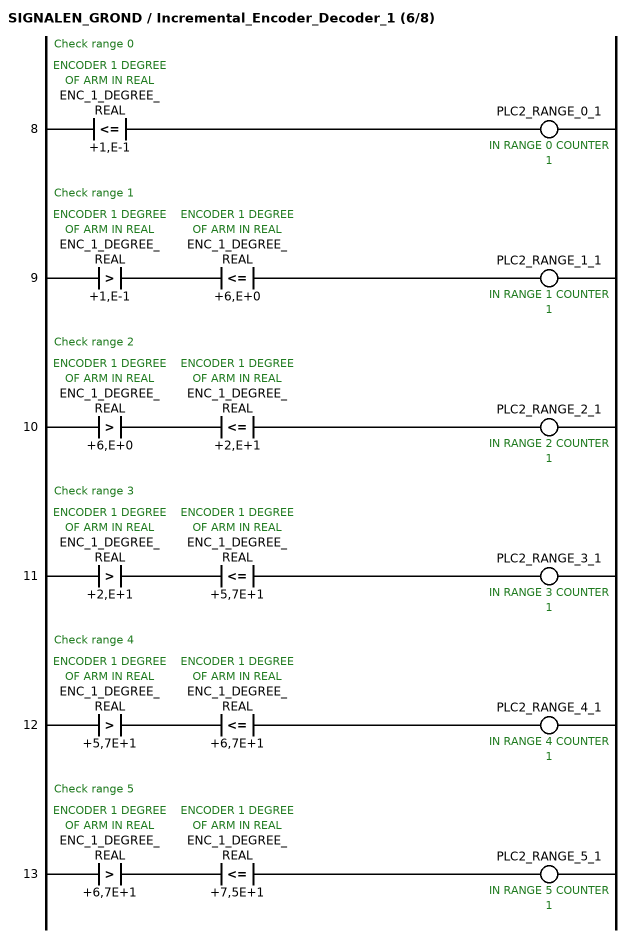
; [picture p325: SIGNALEN_GROND / Incremental_Encoder_Decoder_1, rungs 8-13]
; rung 8: Check range 0
LD<=F(332) ENC_1_DEGREE_REAL +1,E-1  ; ENCODER 1 DEGREE OF ARM IN REAL
OUT PLC2_RANGE_0_1  ; IN RANGE 0 COUNTER 1
; rung 9: Check range 1
LD>F(333) ENC_1_DEGREE_REAL +1,E-1  ; ENCODER 1 DEGREE OF ARM IN REAL
AND<=F(332) ENC_1_DEGREE_REAL +6,E+0  ; ENCODER 1 DEGREE OF ARM IN REAL
OUT PLC2_RANGE_1_1  ; IN RANGE 1 COUNTER 1
; rung 10: Check range 2
LD>F(333) ENC_1_DEGREE_REAL +6,E+0  ; ENCODER 1 DEGREE OF ARM IN REAL
AND<=F(332) ENC_1_DEGREE_REAL +2,E+1  ; ENCODER 1 DEGREE OF ARM IN REAL
OUT PLC2_RANGE_2_1  ; IN RANGE 2 COUNTER 1
; rung 11: Check range 3
LD>F(333) ENC_1_DEGREE_REAL +2,E+1  ; ENCODER 1 DEGREE OF ARM IN REAL
AND<=F(332) ENC_1_DEGREE_REAL +5,7E+1  ; ENCODER 1 DEGREE OF ARM IN REAL
OUT PLC2_RANGE_3_1  ; IN RANGE 3 COUNTER 1
; rung 12: Check range 4
LD>F(333) ENC_1_DEGREE_REAL +5,7E+1  ; ENCODER 1 DEGREE OF ARM IN REAL
AND<=F(332) ENC_1_DEGREE_REAL +6,7E+1  ; ENCODER 1 DEGREE OF ARM IN REAL
OUT PLC2_RANGE_4_1  ; IN RANGE 4 COUNTER 1
; rung 13: Check range 5
LD>F(333) ENC_1_DEGREE_REAL +6,7E+1  ; ENCODER 1 DEGREE OF ARM IN REAL
AND<=F(332) ENC_1_DEGREE_REAL +7,5E+1  ; ENCODER 1 DEGREE OF ARM IN REAL
OUT PLC2_RANGE_5_1  ; IN RANGE 5 COUNTER 1

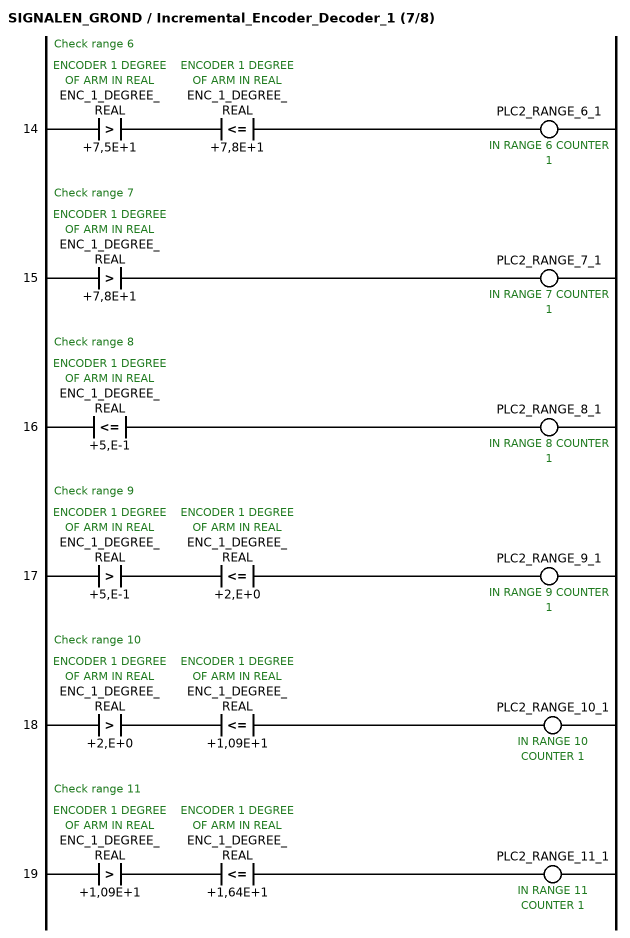
; rung 14: Check range 6
LD>F(333) ENC_1_DEGREE_REAL +7,5E+1  ; ENCODER 1 DEGREE OF ARM IN REAL
AND<=F(332) ENC_1_DEGREE_REAL +7,8E+1  ; ENCODER 1 DEGREE OF ARM IN REAL
OUT PLC2_RANGE_6_1  ; IN RANGE 6 COUNTER 1
; rung 15: Check range 7
LD>F(333) ENC_1_DEGREE_REAL +7,8E+1  ; ENCODER 1 DEGREE OF ARM IN REAL
OUT PLC2_RANGE_7_1  ; IN RANGE 7 COUNTER 1
; rung 16: Check range 8
LD<=F(332) ENC_1_DEGREE_REAL +5,E-1  ; ENCODER 1 DEGREE OF ARM IN REAL
OUT PLC2_RANGE_8_1  ; IN RANGE 8 COUNTER 1
; rung 17: Check range 9
LD>F(333) ENC_1_DEGREE_REAL +5,E-1  ; ENCODER 1 DEGREE OF ARM IN REAL
AND<=F(332) ENC_1_DEGREE_REAL +2,E+0  ; ENCODER 1 DEGREE OF ARM IN REAL
OUT PLC2_RANGE_9_1  ; IN RANGE 9 COUNTER 1
; rung 18: Check range 10
LD>F(333) ENC_1_DEGREE_REAL +2,E+0  ; ENCODER 1 DEGREE OF ARM IN REAL
AND<=F(332) ENC_1_DEGREE_REAL +1,09E+1  ; ENCODER 1 DEGREE OF ARM IN REAL
OUT PLC2_RANGE_10_1  ; IN RANGE 10 COUNTER 1
; rung 19: Check range 11
LD>F(333) ENC_1_DEGREE_REAL +1,09E+1  ; ENCODER 1 DEGREE OF ARM IN REAL
AND<=F(332) ENC_1_DEGREE_REAL +1,64E+1  ; ENCODER 1 DEGREE OF ARM IN REAL
OUT PLC2_RANGE_11_1  ; IN RANGE 11 COUNTER 1

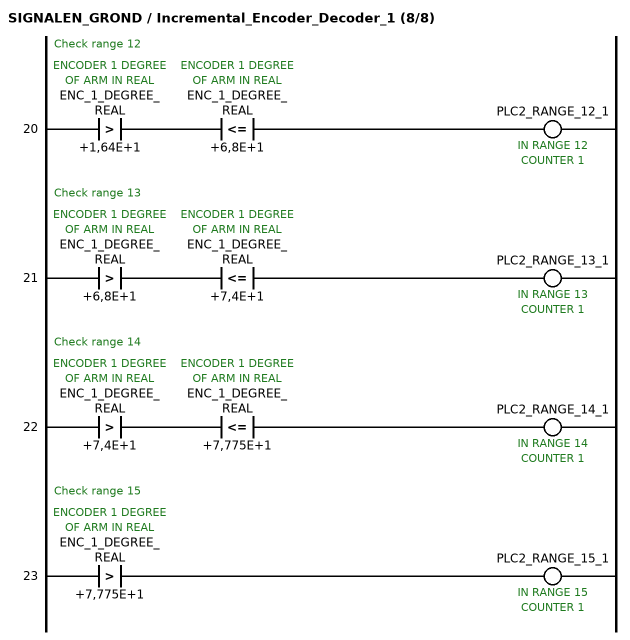
; rung 20: Check range 12
LD>F(333) ENC_1_DEGREE_REAL +1,64E+1  ; ENCODER 1 DEGREE OF ARM IN REAL
AND<=F(332) ENC_1_DEGREE_REAL +6,8E+1  ; ENCODER 1 DEGREE OF ARM IN REAL
OUT PLC2_RANGE_12_1  ; IN RANGE 12 COUNTER 1
; rung 21: Check range 13
LD>F(333) ENC_1_DEGREE_REAL +6,8E+1  ; ENCODER 1 DEGREE OF ARM IN REAL
AND<=F(332) ENC_1_DEGREE_REAL +7,4E+1  ; ENCODER 1 DEGREE OF ARM IN REAL
OUT PLC2_RANGE_13_1  ; IN RANGE 13 COUNTER 1
; rung 22: Check range 14
LD>F(333) ENC_1_DEGREE_REAL +7,4E+1  ; ENCODER 1 DEGREE OF ARM IN REAL
AND<=F(332) ENC_1_DEGREE_REAL +7,775E+1  ; ENCODER 1 DEGREE OF ARM IN REAL
OUT PLC2_RANGE_14_1  ; IN RANGE 14 COUNTER 1
; rung 23: Check range 15
LD>F(333) ENC_1_DEGREE_REAL +7,775E+1  ; ENCODER 1 DEGREE OF ARM IN REAL
OUT PLC2_RANGE_15_1  ; IN RANGE 15 COUNTER 1

### Section Incremental_Encoder_Decoder_2

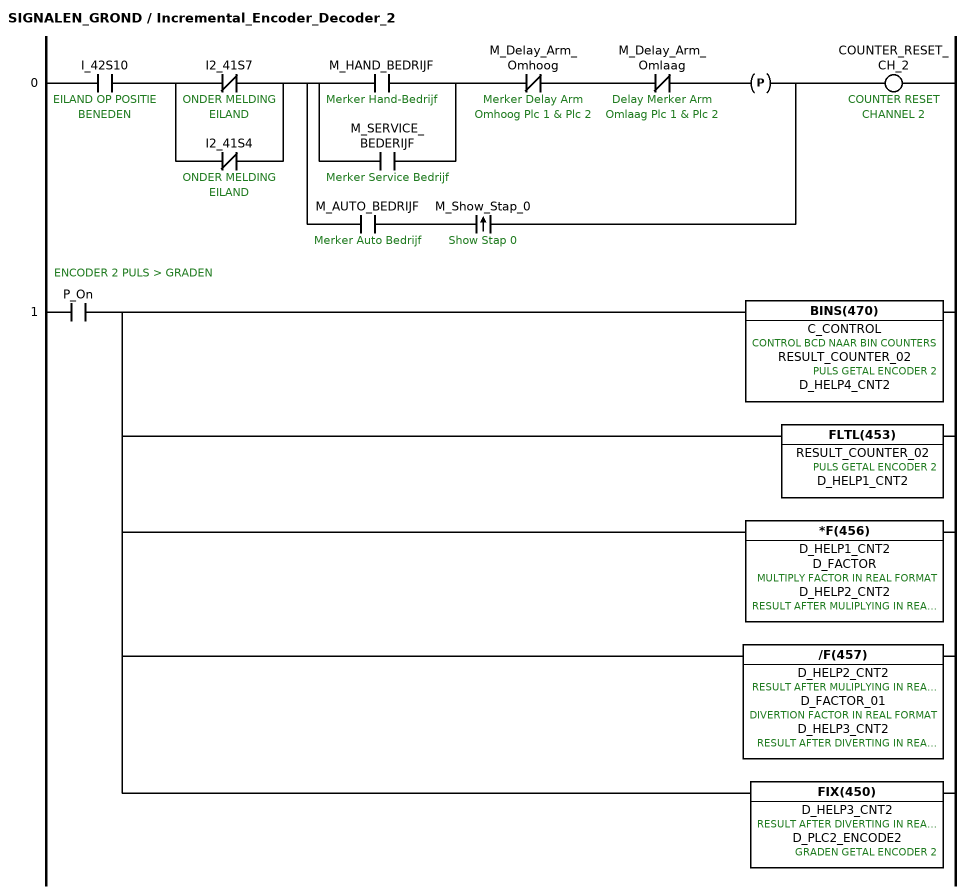
; rung 0
LD I_42S10  ; EILAND OP POSITIE BENEDEN
LDNOT I2_41S7  ; ONDER MELDING EILAND
ORNOT I2_41S4  ; ONDER MELDING EILAND
ANDLD
LD M_HAND_BEDRIJF  ; Merker Hand-Bedrijf
OR M_SERVICE_BEDERIJF  ; Merker Service Bedrijf
ANDNOT M_Delay_Arm_Omhoog  ; Merker Delay Arm Omhoog Plc 1 & Plc 2
ANDNOT M_Delay_Arm_Omlaag  ; Delay Merker Arm Omlaag Plc 1 & Plc 2
UP(521)
LD M_AUTO_BEDRIJF  ; Merker Auto Bedrijf
@AND M_Show_Stap_0  ; Show Stap 0
ORLD
ANDLD
OUT COUNTER_RESET_CH_2  ; COUNTER RESET CHANNEL 2
; rung 1: ENCODER 2 PULS > GRADEN
LD P_On
BINS(470) C_CONTROL RESULT_COUNTER_02 D_HELP4_CNT2  ; CONTROL BCD NAAR BIN COUNTERS, PULS GETAL ENCODER 2
FLTL(453) RESULT_COUNTER_02 D_HELP1_CNT2  ; PULS GETAL ENCODER 2
*F(456) D_HELP1_CNT2 D_FACTOR D_HELP2_CNT2  ; MULTIPLY FACTOR IN REAL FORMAT, RESULT AFTER MULIPLYING IN REAL FORMAT
/F(457) D_HELP2_CNT2 D_FACTOR_01 D_HELP3_CNT2  ; RESULT AFTER MULIPLYING IN REAL FORMAT, DIVERTION FACTOR IN REAL FORMAT, RESULT AFTER DIVERTING IN REAL FORMAT
FIX(450) D_HELP3_CNT2 D_PLC2_ENCODE2  ; RESULT AFTER DIVERTING IN REAL FORMAT, GRADEN GETAL ENCODER 2

### Section Absolute_Encoder_Decoder_3

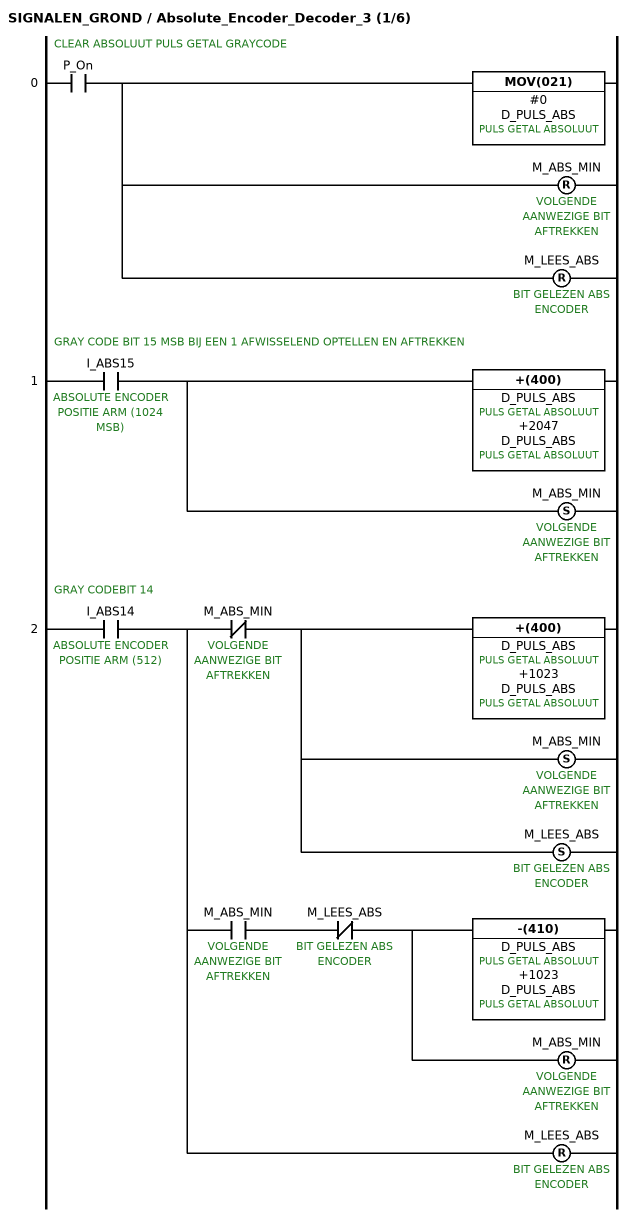
; rung 0: CLEAR ABSOLUUT PULS GETAL GRAYCODE
LD P_On
MOV(021) #0 D_PULS_ABS  ; PULS GETAL ABSOLUUT
RSET M_ABS_MIN  ; VOLGENDE  AANWEZIGE BIT AFTREKKEN
RSET M_LEES_ABS  ; BIT GELEZEN ABS ENCODER
; rung 1: GRAY CODE BIT 15 MSB BIJ EEN 1 AFWISSELEND OPTELLEN EN AFTREKKEN
LD I_ABS15  ; ABSOLUTE ENCODER POSITIE ARM (1024 MSB)
+(400) D_PULS_ABS +2047 D_PULS_ABS  ; PULS GETAL ABSOLUUT
SET M_ABS_MIN  ; VOLGENDE  AANWEZIGE BIT AFTREKKEN
; rung 2: GRAY CODEBIT 14
LD I_ABS14  ; ABSOLUTE ENCODER POSITIE ARM (512)
OUT TR0
ANDNOT M_ABS_MIN  ; VOLGENDE  AANWEZIGE BIT AFTREKKEN
+(400) D_PULS_ABS +1023 D_PULS_ABS  ; PULS GETAL ABSOLUUT
SET M_ABS_MIN  ; VOLGENDE  AANWEZIGE BIT AFTREKKEN
SET M_LEES_ABS  ; BIT GELEZEN ABS ENCODER
LD TR0
AND M_ABS_MIN  ; VOLGENDE  AANWEZIGE BIT AFTREKKEN
ANDNOT M_LEES_ABS  ; BIT GELEZEN ABS ENCODER
-(410) D_PULS_ABS +1023 D_PULS_ABS  ; PULS GETAL ABSOLUUT
RSET M_ABS_MIN  ; VOLGENDE  AANWEZIGE BIT AFTREKKEN
LD TR0
RSET M_LEES_ABS  ; BIT GELEZEN ABS ENCODER

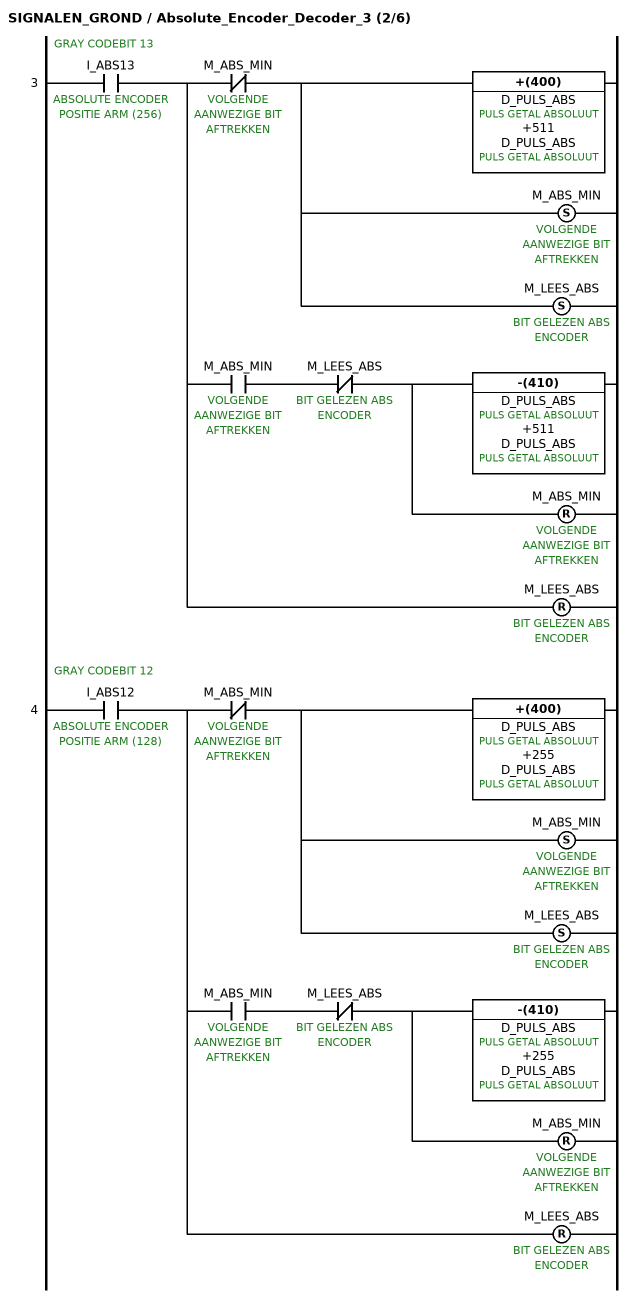
; rung 3: GRAY CODEBIT 13
LD I_ABS13  ; ABSOLUTE ENCODER POSITIE ARM (256)
OUT TR0
ANDNOT M_ABS_MIN  ; VOLGENDE  AANWEZIGE BIT AFTREKKEN
+(400) D_PULS_ABS +511 D_PULS_ABS  ; PULS GETAL ABSOLUUT
SET M_ABS_MIN  ; VOLGENDE  AANWEZIGE BIT AFTREKKEN
SET M_LEES_ABS  ; BIT GELEZEN ABS ENCODER
LD TR0
AND M_ABS_MIN  ; VOLGENDE  AANWEZIGE BIT AFTREKKEN
ANDNOT M_LEES_ABS  ; BIT GELEZEN ABS ENCODER
-(410) D_PULS_ABS +511 D_PULS_ABS  ; PULS GETAL ABSOLUUT
RSET M_ABS_MIN  ; VOLGENDE  AANWEZIGE BIT AFTREKKEN
LD TR0
RSET M_LEES_ABS  ; BIT GELEZEN ABS ENCODER
; rung 4: GRAY CODEBIT 12
LD I_ABS12  ; ABSOLUTE ENCODER POSITIE ARM (128)
OUT TR0
ANDNOT M_ABS_MIN  ; VOLGENDE  AANWEZIGE BIT AFTREKKEN
+(400) D_PULS_ABS +255 D_PULS_ABS  ; PULS GETAL ABSOLUUT
SET M_ABS_MIN  ; VOLGENDE  AANWEZIGE BIT AFTREKKEN
SET M_LEES_ABS  ; BIT GELEZEN ABS ENCODER
LD TR0
AND M_ABS_MIN  ; VOLGENDE  AANWEZIGE BIT AFTREKKEN
ANDNOT M_LEES_ABS  ; BIT GELEZEN ABS ENCODER
-(410) D_PULS_ABS +255 D_PULS_ABS  ; PULS GETAL ABSOLUUT
RSET M_ABS_MIN  ; VOLGENDE  AANWEZIGE BIT AFTREKKEN
LD TR0
RSET M_LEES_ABS  ; BIT GELEZEN ABS ENCODER

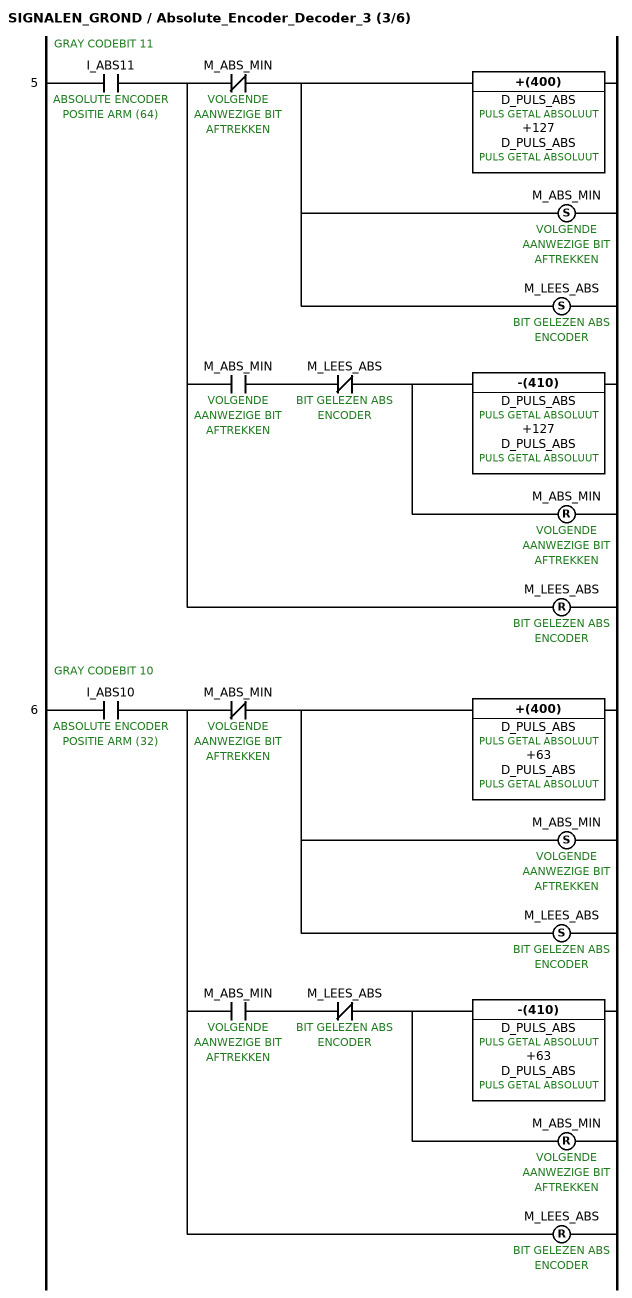
; rung 5: GRAY CODEBIT 11
LD I_ABS11  ; ABSOLUTE ENCODER POSITIE ARM (64)
OUT TR0
ANDNOT M_ABS_MIN  ; VOLGENDE  AANWEZIGE BIT AFTREKKEN
+(400) D_PULS_ABS +127 D_PULS_ABS  ; PULS GETAL ABSOLUUT
SET M_ABS_MIN  ; VOLGENDE  AANWEZIGE BIT AFTREKKEN
SET M_LEES_ABS  ; BIT GELEZEN ABS ENCODER
LD TR0
AND M_ABS_MIN  ; VOLGENDE  AANWEZIGE BIT AFTREKKEN
ANDNOT M_LEES_ABS  ; BIT GELEZEN ABS ENCODER
-(410) D_PULS_ABS +127 D_PULS_ABS  ; PULS GETAL ABSOLUUT
RSET M_ABS_MIN  ; VOLGENDE  AANWEZIGE BIT AFTREKKEN
LD TR0
RSET M_LEES_ABS  ; BIT GELEZEN ABS ENCODER
; rung 6: GRAY CODEBIT 10
LD I_ABS10  ; ABSOLUTE ENCODER POSITIE ARM (32)
OUT TR0
ANDNOT M_ABS_MIN  ; VOLGENDE  AANWEZIGE BIT AFTREKKEN
+(400) D_PULS_ABS +63 D_PULS_ABS  ; PULS GETAL ABSOLUUT
SET M_ABS_MIN  ; VOLGENDE  AANWEZIGE BIT AFTREKKEN
SET M_LEES_ABS  ; BIT GELEZEN ABS ENCODER
LD TR0
AND M_ABS_MIN  ; VOLGENDE  AANWEZIGE BIT AFTREKKEN
ANDNOT M_LEES_ABS  ; BIT GELEZEN ABS ENCODER
-(410) D_PULS_ABS +63 D_PULS_ABS  ; PULS GETAL ABSOLUUT
RSET M_ABS_MIN  ; VOLGENDE  AANWEZIGE BIT AFTREKKEN
LD TR0
RSET M_LEES_ABS  ; BIT GELEZEN ABS ENCODER

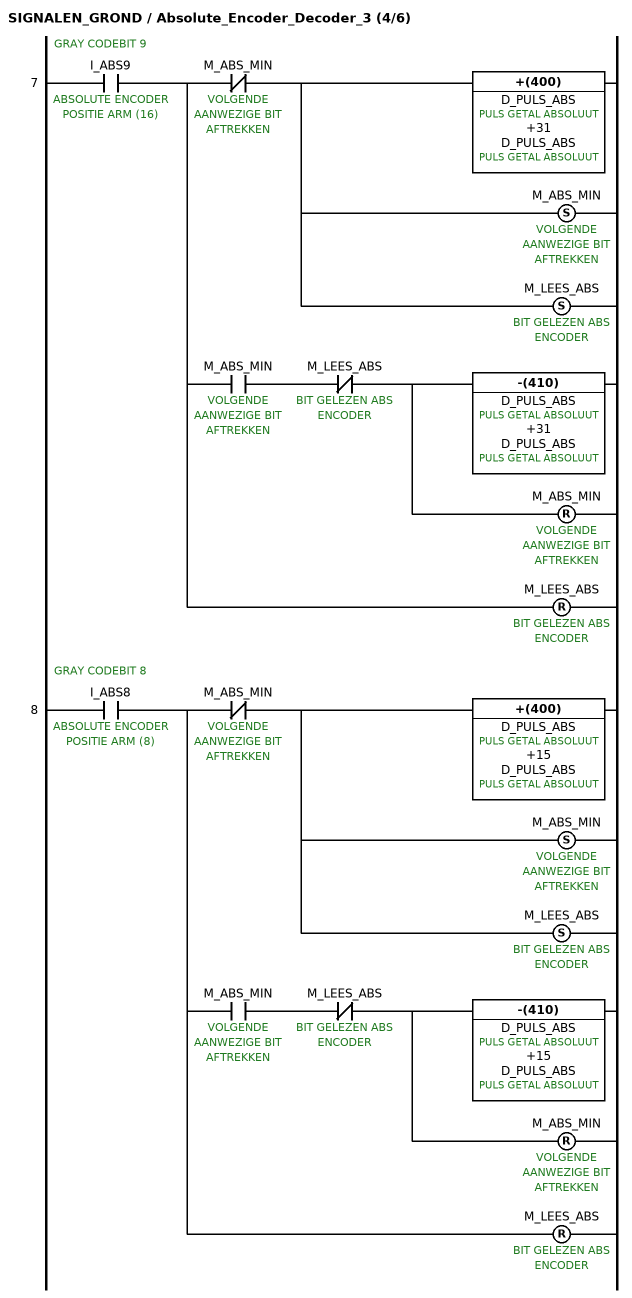
; rung 7: GRAY CODEBIT 9
LD I_ABS9  ; ABSOLUTE ENCODER POSITIE ARM (16)
OUT TR0
ANDNOT M_ABS_MIN  ; VOLGENDE  AANWEZIGE BIT AFTREKKEN
+(400) D_PULS_ABS +31 D_PULS_ABS  ; PULS GETAL ABSOLUUT
SET M_ABS_MIN  ; VOLGENDE  AANWEZIGE BIT AFTREKKEN
SET M_LEES_ABS  ; BIT GELEZEN ABS ENCODER
LD TR0
AND M_ABS_MIN  ; VOLGENDE  AANWEZIGE BIT AFTREKKEN
ANDNOT M_LEES_ABS  ; BIT GELEZEN ABS ENCODER
-(410) D_PULS_ABS +31 D_PULS_ABS  ; PULS GETAL ABSOLUUT
RSET M_ABS_MIN  ; VOLGENDE  AANWEZIGE BIT AFTREKKEN
LD TR0
RSET M_LEES_ABS  ; BIT GELEZEN ABS ENCODER
; rung 8: GRAY CODEBIT 8
LD I_ABS8  ; ABSOLUTE ENCODER POSITIE ARM (8)
OUT TR0
ANDNOT M_ABS_MIN  ; VOLGENDE  AANWEZIGE BIT AFTREKKEN
+(400) D_PULS_ABS +15 D_PULS_ABS  ; PULS GETAL ABSOLUUT
SET M_ABS_MIN  ; VOLGENDE  AANWEZIGE BIT AFTREKKEN
SET M_LEES_ABS  ; BIT GELEZEN ABS ENCODER
LD TR0
AND M_ABS_MIN  ; VOLGENDE  AANWEZIGE BIT AFTREKKEN
ANDNOT M_LEES_ABS  ; BIT GELEZEN ABS ENCODER
-(410) D_PULS_ABS +15 D_PULS_ABS  ; PULS GETAL ABSOLUUT
RSET M_ABS_MIN  ; VOLGENDE  AANWEZIGE BIT AFTREKKEN
LD TR0
RSET M_LEES_ABS  ; BIT GELEZEN ABS ENCODER

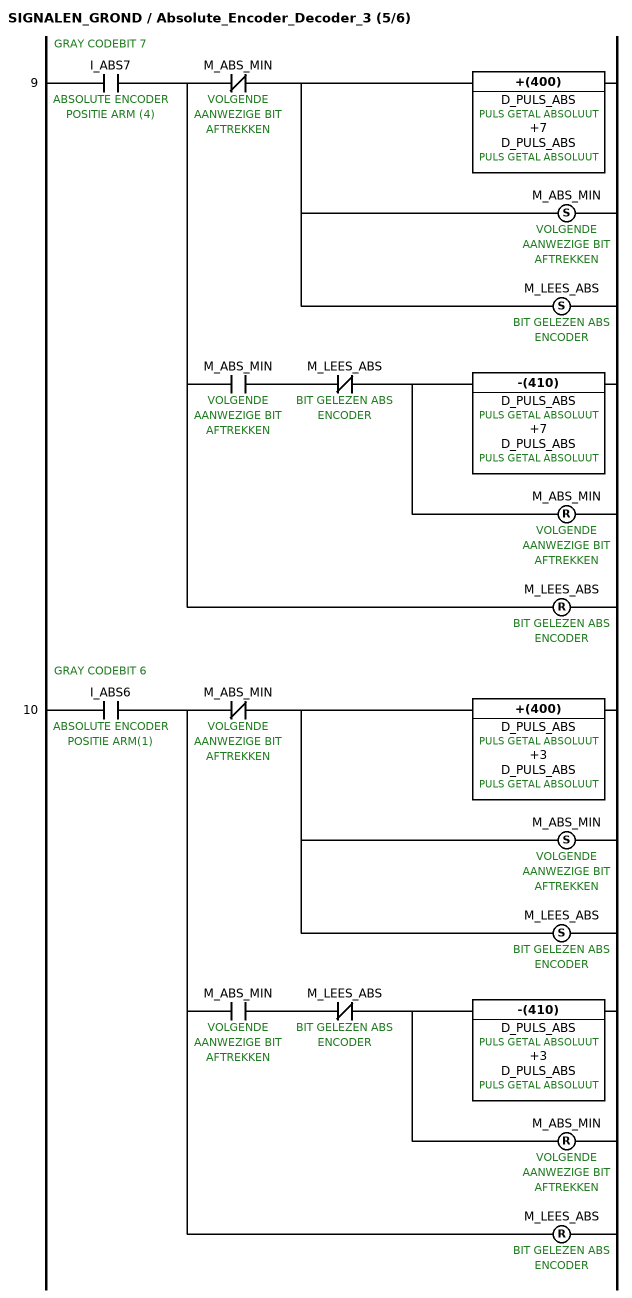
; rung 9: GRAY CODEBIT 7
LD I_ABS7  ; ABSOLUTE ENCODER POSITIE ARM (4)
OUT TR0
ANDNOT M_ABS_MIN  ; VOLGENDE  AANWEZIGE BIT AFTREKKEN
+(400) D_PULS_ABS +7 D_PULS_ABS  ; PULS GETAL ABSOLUUT
SET M_ABS_MIN  ; VOLGENDE  AANWEZIGE BIT AFTREKKEN
SET M_LEES_ABS  ; BIT GELEZEN ABS ENCODER
LD TR0
AND M_ABS_MIN  ; VOLGENDE  AANWEZIGE BIT AFTREKKEN
ANDNOT M_LEES_ABS  ; BIT GELEZEN ABS ENCODER
-(410) D_PULS_ABS +7 D_PULS_ABS  ; PULS GETAL ABSOLUUT
RSET M_ABS_MIN  ; VOLGENDE  AANWEZIGE BIT AFTREKKEN
LD TR0
RSET M_LEES_ABS  ; BIT GELEZEN ABS ENCODER
; rung 10: GRAY CODEBIT 6
LD I_ABS6  ; ABSOLUTE ENCODER POSITIE ARM(1)
OUT TR0
ANDNOT M_ABS_MIN  ; VOLGENDE  AANWEZIGE BIT AFTREKKEN
+(400) D_PULS_ABS +3 D_PULS_ABS  ; PULS GETAL ABSOLUUT
SET M_ABS_MIN  ; VOLGENDE  AANWEZIGE BIT AFTREKKEN
SET M_LEES_ABS  ; BIT GELEZEN ABS ENCODER
LD TR0
AND M_ABS_MIN  ; VOLGENDE  AANWEZIGE BIT AFTREKKEN
ANDNOT M_LEES_ABS  ; BIT GELEZEN ABS ENCODER
-(410) D_PULS_ABS +3 D_PULS_ABS  ; PULS GETAL ABSOLUUT
RSET M_ABS_MIN  ; VOLGENDE  AANWEZIGE BIT AFTREKKEN
LD TR0
RSET M_LEES_ABS  ; BIT GELEZEN ABS ENCODER

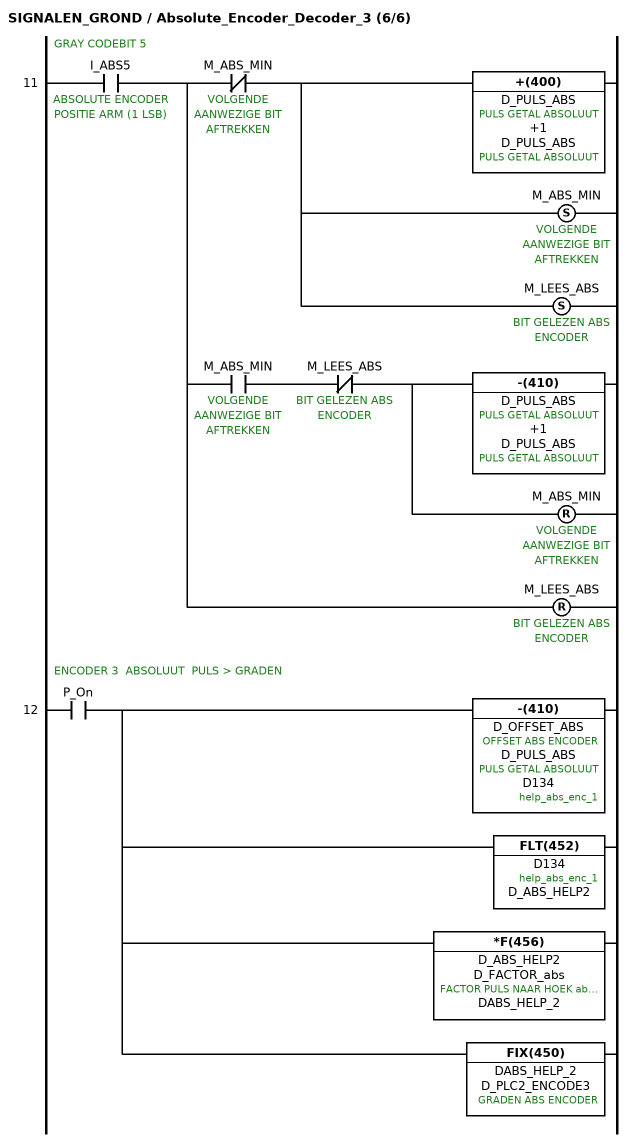
; rung 11: GRAY CODEBIT 5
LD I_ABS5  ; ABSOLUTE ENCODER POSITIE ARM (1 LSB)
OUT TR0
ANDNOT M_ABS_MIN  ; VOLGENDE  AANWEZIGE BIT AFTREKKEN
+(400) D_PULS_ABS +1 D_PULS_ABS  ; PULS GETAL ABSOLUUT
SET M_ABS_MIN  ; VOLGENDE  AANWEZIGE BIT AFTREKKEN
SET M_LEES_ABS  ; BIT GELEZEN ABS ENCODER
LD TR0
AND M_ABS_MIN  ; VOLGENDE  AANWEZIGE BIT AFTREKKEN
ANDNOT M_LEES_ABS  ; BIT GELEZEN ABS ENCODER
-(410) D_PULS_ABS +1 D_PULS_ABS  ; PULS GETAL ABSOLUUT
RSET M_ABS_MIN  ; VOLGENDE  AANWEZIGE BIT AFTREKKEN
LD TR0
RSET M_LEES_ABS  ; BIT GELEZEN ABS ENCODER
; rung 12: ENCODER 3  ABSOLUUT  PULS > GRADEN
LD P_On
-(410) D_OFFSET_ABS D_PULS_ABS D134  ; OFFSET ABS ENCODER, PULS GETAL ABSOLUUT, help_abs_enc_1
FLT(452) D134 D_ABS_HELP2  ; help_abs_enc_1
*F(456) D_ABS_HELP2 D_FACTOR_abs DABS_HELP_2  ; FACTOR PULS NAAR HOEK abs encoder
FIX(450) DABS_HELP_2 D_PLC2_ENCODE3  ; GRADEN ABS ENCODER

### Section Controle_Positie_Arm

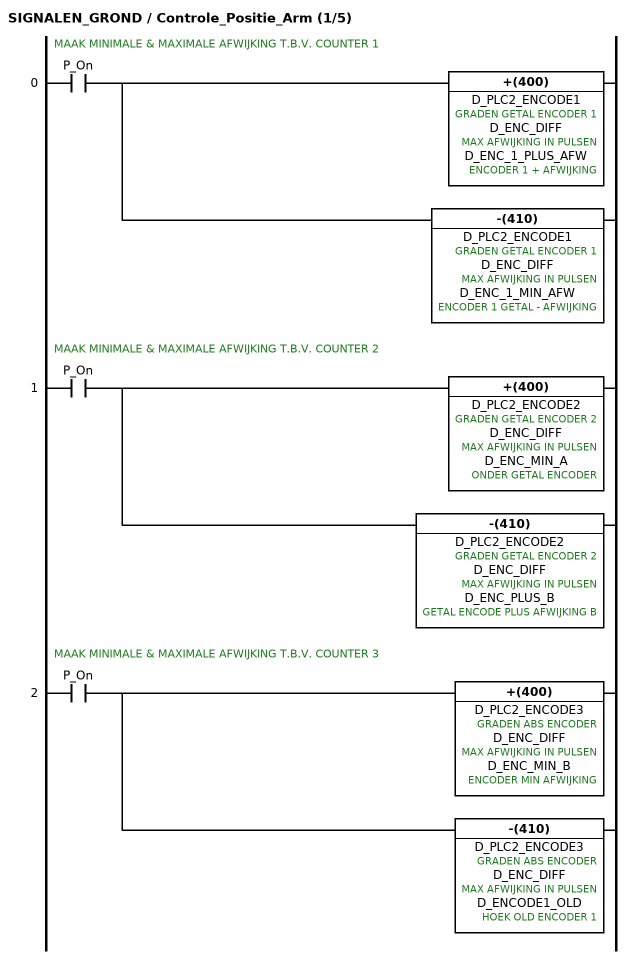
; rung 0: MAAK MINIMALE & MAXIMALE AFWIJKING T.B.V. COUNTER 1
LD P_On
+(400) D_PLC2_ENCODE1 D_ENC_DIFF D_ENC_1_PLUS_AFW  ; GRADEN GETAL ENCODER 1, MAX AFWIJKING IN PULSEN, ENCODER 1 + AFWIJKING
-(410) D_PLC2_ENCODE1 D_ENC_DIFF D_ENC_1_MIN_AFW  ; GRADEN GETAL ENCODER 1, MAX AFWIJKING IN PULSEN, ENCODER 1 GETAL - AFWIJKING
; rung 1: MAAK MINIMALE & MAXIMALE AFWIJKING T.B.V. COUNTER 2
LD P_On
+(400) D_PLC2_ENCODE2 D_ENC_DIFF D_ENC_MIN_A  ; GRADEN GETAL ENCODER 2, MAX AFWIJKING IN PULSEN, ONDER GETAL ENCODER
-(410) D_PLC2_ENCODE2 D_ENC_DIFF D_ENC_PLUS_B  ; GRADEN GETAL ENCODER 2, MAX AFWIJKING IN PULSEN, GETAL ENCODE PLUS AFWIJKING B
; rung 2: MAAK MINIMALE & MAXIMALE AFWIJKING T.B.V. COUNTER 3
LD P_On
+(400) D_PLC2_ENCODE3 D_ENC_DIFF D_ENC_MIN_B  ; GRADEN ABS ENCODER, MAX AFWIJKING IN PULSEN, ENCODER MIN AFWIJKING
-(410) D_PLC2_ENCODE3 D_ENC_DIFF D_ENCODE1_OLD  ; GRADEN ABS ENCODER, MAX AFWIJKING IN PULSEN, HOEK OLD ENCODER 1

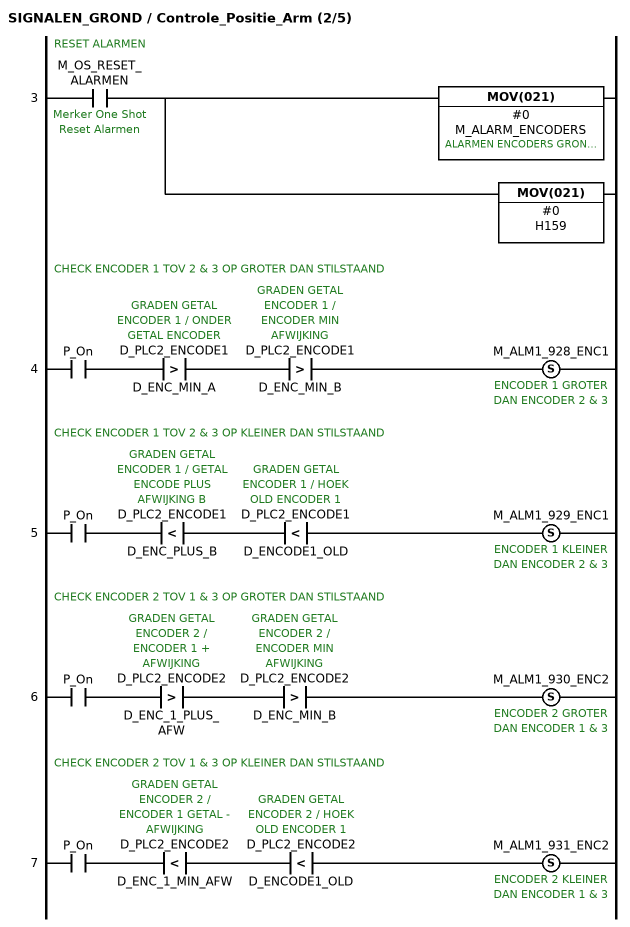
; rung 3: RESET ALARMEN
LD M_OS_RESET_ALARMEN  ; Merker One Shot Reset Alarmen
MOV(021) #0 M_ALARM_ENCODERS  ; ALARMEN ENCODERS GROND 928-943
MOV(021) #0 H159
; rung 4: CHECK ENCODER 1 TOV 2 & 3 OP GROTER DAN STILSTAAND
LD P_On
AND>S(322) D_PLC2_ENCODE1 D_ENC_MIN_A  ; GRADEN GETAL ENCODER 1, ONDER GETAL ENCODER
AND>S(322) D_PLC2_ENCODE1 D_ENC_MIN_B  ; GRADEN GETAL ENCODER 1, ENCODER MIN AFWIJKING
SET M_ALM1_928_ENC1  ; ENCODER 1 GROTER DAN ENCODER 2 & 3
; rung 5: CHECK ENCODER 1 TOV 2 & 3 OP KLEINER DAN STILSTAAND
LD P_On
AND<S(312) D_PLC2_ENCODE1 D_ENC_PLUS_B  ; GRADEN GETAL ENCODER 1, GETAL ENCODE PLUS AFWIJKING B
AND<S(312) D_PLC2_ENCODE1 D_ENCODE1_OLD  ; GRADEN GETAL ENCODER 1, HOEK OLD ENCODER 1
SET M_ALM1_929_ENC1  ; ENCODER 1 KLEINER DAN ENCODER 2 & 3
; rung 6: CHECK ENCODER 2 TOV 1 & 3 OP GROTER DAN STILSTAAND
LD P_On
AND>S(322) D_PLC2_ENCODE2 D_ENC_1_PLUS_AFW  ; GRADEN GETAL ENCODER 2, ENCODER 1 + AFWIJKING
AND>S(322) D_PLC2_ENCODE2 D_ENC_MIN_B  ; GRADEN GETAL ENCODER 2, ENCODER MIN AFWIJKING
SET M_ALM1_930_ENC2  ; ENCODER 2 GROTER DAN ENCODER 1 & 3
; rung 7: CHECK ENCODER 2 TOV 1 & 3 OP KLEINER DAN STILSTAAND
LD P_On
AND<S(312) D_PLC2_ENCODE2 D_ENC_1_MIN_AFW  ; GRADEN GETAL ENCODER 2, ENCODER 1 GETAL - AFWIJKING
AND<S(312) D_PLC2_ENCODE2 D_ENCODE1_OLD  ; GRADEN GETAL ENCODER 2, HOEK OLD ENCODER 1
SET M_ALM1_931_ENC2  ; ENCODER 2 KLEINER DAN ENCODER 1 & 3

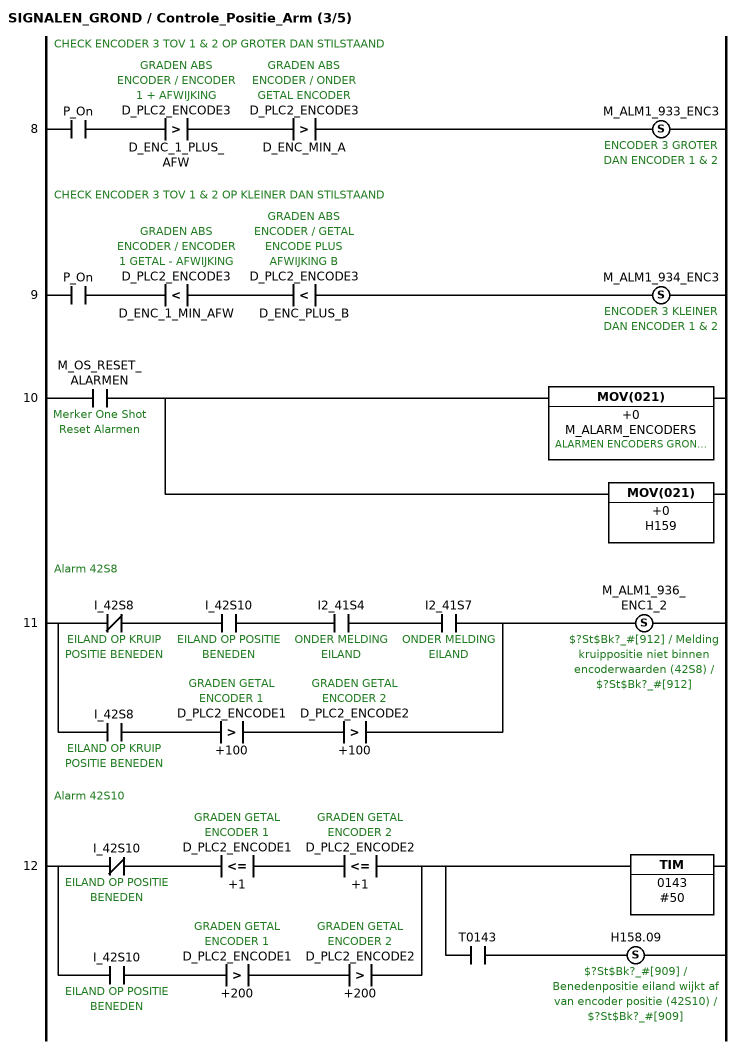
; rung 8: CHECK ENCODER 3 TOV 1 & 2 OP GROTER DAN STILSTAAND
LD P_On
AND>S(322) D_PLC2_ENCODE3 D_ENC_1_PLUS_AFW  ; GRADEN ABS ENCODER, ENCODER 1 + AFWIJKING
AND>S(322) D_PLC2_ENCODE3 D_ENC_MIN_A  ; GRADEN ABS ENCODER, ONDER GETAL ENCODER
SET M_ALM1_933_ENC3  ; ENCODER 3 GROTER DAN ENCODER 1 & 2
; rung 9: CHECK ENCODER 3 TOV 1 & 2 OP KLEINER DAN STILSTAAND
LD P_On
AND<S(312) D_PLC2_ENCODE3 D_ENC_1_MIN_AFW  ; GRADEN ABS ENCODER, ENCODER 1 GETAL - AFWIJKING
AND<S(312) D_PLC2_ENCODE3 D_ENC_PLUS_B  ; GRADEN ABS ENCODER, GETAL ENCODE PLUS AFWIJKING B
SET M_ALM1_934_ENC3  ; ENCODER 3 KLEINER DAN ENCODER 1 & 2
; rung 10
LD M_OS_RESET_ALARMEN  ; Merker One Shot Reset Alarmen
MOV(021) +0 M_ALARM_ENCODERS  ; ALARMEN ENCODERS GROND 928-943
MOV(021) +0 H159
; rung 11: Alarm 42S8
LDNOT I_42S8  ; EILAND OP KRUIP POSITIE BENEDEN
AND I_42S10  ; EILAND OP POSITIE BENEDEN
AND I2_41S4  ; ONDER MELDING EILAND
AND I2_41S7  ; ONDER MELDING EILAND
LD I_42S8  ; EILAND OP KRUIP POSITIE BENEDEN
AND>S(322) D_PLC2_ENCODE1 +100  ; GRADEN GETAL ENCODER 1
AND>S(322) D_PLC2_ENCODE2 +100  ; GRADEN GETAL ENCODER 2
ORLD
SET M_ALM1_936_ENC1_2  ; $?St$Bk?_#[912] / Melding kruippositie niet binnen encoderwaarden (42S8) / $?St$Bk?_#[912]
; rung 12: Alarm 42S10
LDNOT I_42S10  ; EILAND OP POSITIE BENEDEN
AND<=S(317) D_PLC2_ENCODE1 +1  ; GRADEN GETAL ENCODER 1
AND<=S(317) D_PLC2_ENCODE2 +1  ; GRADEN GETAL ENCODER 2
LD I_42S10  ; EILAND OP POSITIE BENEDEN
AND>S(322) D_PLC2_ENCODE1 +200  ; GRADEN GETAL ENCODER 1
AND>S(322) D_PLC2_ENCODE2 +200  ; GRADEN GETAL ENCODER 2
ORLD
TIM 0143 #50
AND T0143
SET H158.09  ; $?St$Bk?_#[909] / Benedenpositie eiland wijkt af van encoder positie (42S10) / $?St$Bk?_#[909]

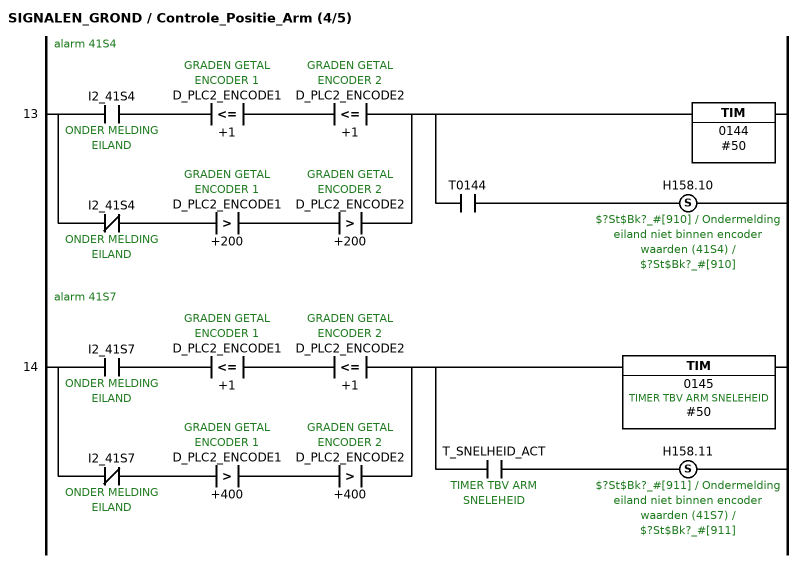
; rung 13: alarm 41S4
LD I2_41S4  ; ONDER MELDING EILAND
AND<=S(317) D_PLC2_ENCODE1 +1  ; GRADEN GETAL ENCODER 1
AND<=S(317) D_PLC2_ENCODE2 +1  ; GRADEN GETAL ENCODER 2
LDNOT I2_41S4  ; ONDER MELDING EILAND
AND>S(322) D_PLC2_ENCODE1 +200  ; GRADEN GETAL ENCODER 1
AND>S(322) D_PLC2_ENCODE2 +200  ; GRADEN GETAL ENCODER 2
ORLD
TIM 0144 #50
AND T0144
SET H158.10  ; $?St$Bk?_#[910] / Ondermelding eiland niet binnen encoder waarden (41S4) / $?St$Bk?_#[910]
; rung 14: alarm 41S7
LD I2_41S7  ; ONDER MELDING EILAND
AND<=S(317) D_PLC2_ENCODE1 +1  ; GRADEN GETAL ENCODER 1
AND<=S(317) D_PLC2_ENCODE2 +1  ; GRADEN GETAL ENCODER 2
LDNOT I2_41S7  ; ONDER MELDING EILAND
AND>S(322) D_PLC2_ENCODE1 +400  ; GRADEN GETAL ENCODER 1
AND>S(322) D_PLC2_ENCODE2 +400  ; GRADEN GETAL ENCODER 2
ORLD
TIM 0145 #50  ; TIMER TBV ARM SNELEHEID
AND T_SNELHEID_ACT  ; TIMER TBV ARM SNELEHEID
SET H158.11  ; $?St$Bk?_#[911] / Ondermelding eiland niet binnen encoder waarden (41S7) / $?St$Bk?_#[911]

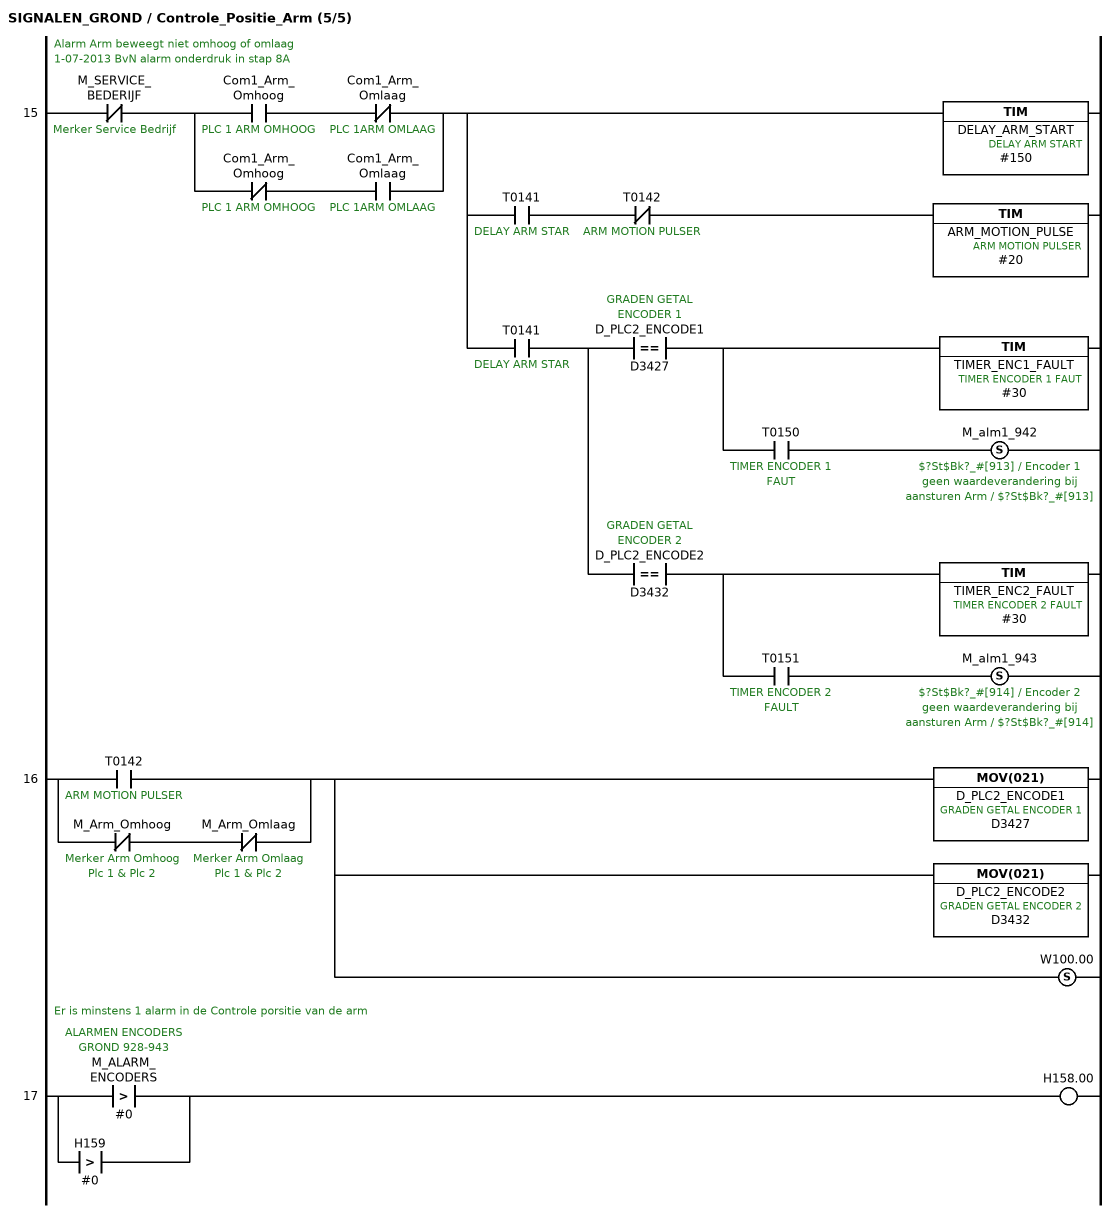
; rung 15: Alarm Arm beweegt niet omhoog of omlaag / 1-07-2013 BvN alarm onderdruk in stap 8A
LDNOT M_SERVICE_BEDERIJF  ; Merker Service Bedrijf
LD Com1_Arm_Omhoog  ; PLC 1 ARM OMHOOG
ANDNOT Com1_Arm_Omlaag  ; PLC 1ARM OMLAAG
LDNOT Com1_Arm_Omhoog  ; PLC 1 ARM OMHOOG
AND Com1_Arm_Omlaag  ; PLC 1ARM OMLAAG
ORLD
ANDLD
OUT TR0
TIM DELAY_ARM_START #150  ; DELAY ARM START
AND T0141  ; DELAY ARM STAR
ANDNOT T0142  ; ARM MOTION PULSER
TIM ARM_MOTION_PULSE #20  ; ARM MOTION PULSER
LD TR0
AND T0141  ; DELAY ARM STAR
OUT TR0
AND=(300) D_PLC2_ENCODE1 D3427  ; GRADEN GETAL ENCODER 1
TIM TIMER_ENC1_FAULT #30  ; TIMER ENCODER 1 FAUT
AND T0150  ; TIMER ENCODER 1 FAUT
SET M_alm1_942  ; $?St$Bk?_#[913] / Encoder 1 geen waardeverandering bij aansturen Arm / $?St$Bk?_#[913]
LD TR0
AND=(300) D_PLC2_ENCODE2 D3432  ; GRADEN GETAL ENCODER 2
TIM TIMER_ENC2_FAULT #30  ; TIMER ENCODER 2 FAULT
AND T0151  ; TIMER ENCODER 2 FAULT
SET M_alm1_943  ; $?St$Bk?_#[914] / Encoder 2 geen waardeverandering bij aansturen Arm / $?St$Bk?_#[914]
; rung 16
LD T0142  ; ARM MOTION PULSER
LDNOT M_Arm_Omhoog  ; Merker Arm Omhoog Plc 1 & Plc 2
ANDNOT M_Arm_Omlaag  ; Merker Arm Omlaag Plc 1 & Plc 2
ORLD
MOV(021) D_PLC2_ENCODE1 D3427  ; GRADEN GETAL ENCODER 1
MOV(021) D_PLC2_ENCODE2 D3432  ; GRADEN GETAL ENCODER 2
SET W100.00
; rung 17: Er is minstens 1 alarm in de Controle porsitie van de arm
LD>(320) M_ALARM_ENCODERS #0  ; ALARMEN ENCODERS GROND 928-943
OR>(320) H159 #0
OUT H158.00

### Section Controle_Snelheid_Arm

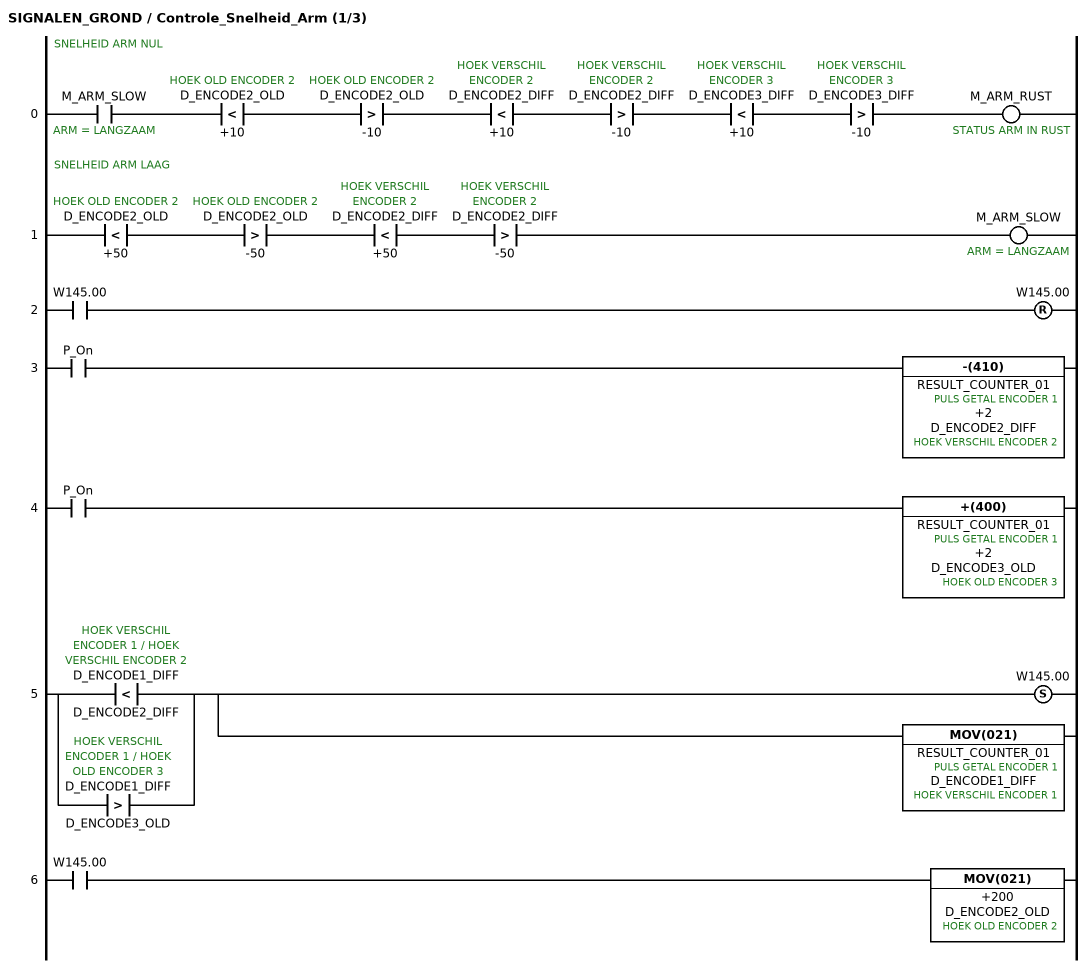
; rung 0: SNELHEID ARM NUL
LD M_ARM_SLOW  ; ARM = LANGZAAM
AND<S(312) D_ENCODE2_OLD +10  ; HOEK OLD ENCODER 2
AND>S(322) D_ENCODE2_OLD -10  ; HOEK OLD ENCODER 2
AND<S(312) D_ENCODE2_DIFF +10  ; HOEK VERSCHIL ENCODER 2
AND>S(322) D_ENCODE2_DIFF -10  ; HOEK VERSCHIL ENCODER 2
AND<S(312) D_ENCODE3_DIFF +10  ; HOEK VERSCHIL ENCODER 3
AND>S(322) D_ENCODE3_DIFF -10  ; HOEK VERSCHIL ENCODER 3
OUT M_ARM_RUST  ; STATUS ARM IN RUST
; rung 1: SNELHEID ARM LAAG
LD<S(312) D_ENCODE2_OLD +50  ; HOEK OLD ENCODER 2
AND>S(322) D_ENCODE2_OLD -50  ; HOEK OLD ENCODER 2
AND<S(312) D_ENCODE2_DIFF +50  ; HOEK VERSCHIL ENCODER 2
AND>S(322) D_ENCODE2_DIFF -50  ; HOEK VERSCHIL ENCODER 2
OUT M_ARM_SLOW  ; ARM = LANGZAAM
; rung 2
LD W145.00
RSET W145.00
; rung 3
LD P_On
-(410) RESULT_COUNTER_01 +2 D_ENCODE2_DIFF  ; PULS GETAL ENCODER 1, HOEK VERSCHIL ENCODER 2
; rung 4
LD P_On
+(400) RESULT_COUNTER_01 +2 D_ENCODE3_OLD  ; PULS GETAL ENCODER 1, HOEK OLD ENCODER 3
; rung 5
LD<(310) D_ENCODE1_DIFF D_ENCODE2_DIFF  ; HOEK VERSCHIL ENCODER 1, HOEK VERSCHIL ENCODER 2
OR>(320) D_ENCODE1_DIFF D_ENCODE3_OLD  ; HOEK VERSCHIL ENCODER 1, HOEK OLD ENCODER 3
SET W145.00
MOV(021) RESULT_COUNTER_01 D_ENCODE1_DIFF  ; PULS GETAL ENCODER 1, HOEK VERSCHIL ENCODER 1
; rung 6
LD W145.00
MOV(021) +200 D_ENCODE2_OLD  ; HOEK OLD ENCODER 2

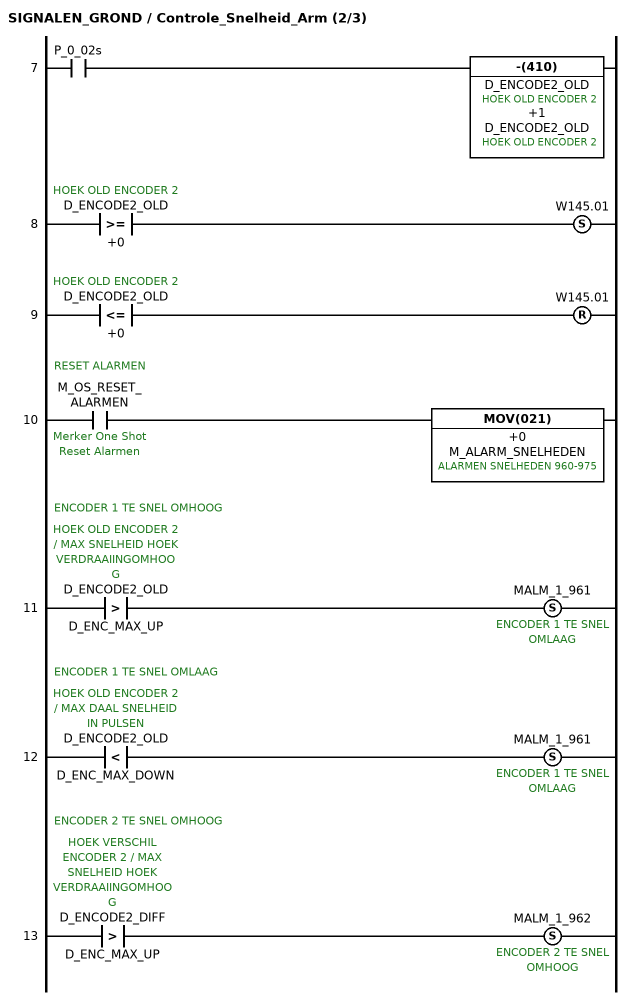
; rung 7
LD P_0_02s
-(410) D_ENCODE2_OLD +1 D_ENCODE2_OLD  ; HOEK OLD ENCODER 2
; rung 8
LD>=S(327) D_ENCODE2_OLD +0  ; HOEK OLD ENCODER 2
SET W145.01
; rung 9
LD<=S(317) D_ENCODE2_OLD +0  ; HOEK OLD ENCODER 2
RSET W145.01
; rung 10: RESET ALARMEN
LD M_OS_RESET_ALARMEN  ; Merker One Shot Reset Alarmen
MOV(021) +0 M_ALARM_SNELHEDEN  ; ALARMEN SNELHEDEN 960-975
; rung 11: ENCODER 1 TE SNEL OMHOOG
LD>S(322) D_ENCODE2_OLD D_ENC_MAX_UP  ; HOEK OLD ENCODER 2, MAX SNELHEID HOEK VERDRAAIINGOMHOOG
SET MALM_1_961  ; ENCODER 1 TE SNEL OMLAAG
; rung 12: ENCODER 1 TE SNEL OMLAAG
LD<S(312) D_ENCODE2_OLD D_ENC_MAX_DOWN  ; HOEK OLD ENCODER 2, MAX DAAL SNELHEID IN PULSEN
SET MALM_1_961  ; ENCODER 1 TE SNEL OMLAAG
; rung 13: ENCODER 2 TE SNEL OMHOOG
LD>S(322) D_ENCODE2_DIFF D_ENC_MAX_UP  ; HOEK VERSCHIL ENCODER 2, MAX SNELHEID HOEK VERDRAAIINGOMHOOG
SET MALM_1_962  ; ENCODER 2 TE SNEL OMHOOG

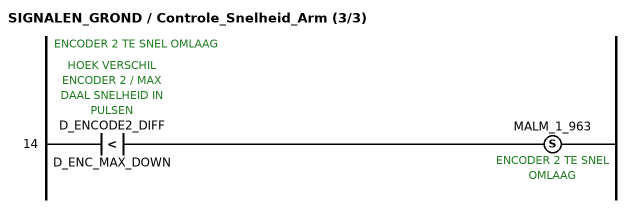
; rung 14: ENCODER 2 TE SNEL OMLAAG
LD<S(312) D_ENCODE2_DIFF D_ENC_MAX_DOWN  ; HOEK VERSCHIL ENCODER 2, MAX DAAL SNELHEID IN PULSEN
SET MALM_1_963  ; ENCODER 2 TE SNEL OMLAAG

### Section Einde_Signalering_Grond
; rung 0
END(001)

## Program BESTURING_GROND (cyclic task 6)
Local symbols
Com1_Alle_Oever_Poortjes_Gesloten 3032.15 BOOL  ; Alle Oever Poortjes zijn gesloten
Com1_Ingangs_Poortje_1_Links_Open 3032.01 BOOL
Com1_Open_Ingangs_Poort_1_L 3032.03 BOOL
Com1_Open_Uitgangs_Poortjes 3033.03 BOOL  ; Open de Uitgangs Poortjes
Com1_Sluit_Uitgangs_Poortjes_Oever 3033.04 BOOL  ; Sluit de Uitgangs Poortjes Oever
Com1_Vrijgave_Ingangs_Poortjes 3032.01 BOOL
Com2_Act_Groter_Snelheid 3337.04 BOOL  ; Actuele snelheid groter dan wens snelheid
Com2_Act_Kleiner_Snelheid 3337.06 BOOL  ; Actuele snelheid kleiner dan wens snelheid
Com2_Act_gelijk_Snelheid 3337.05 BOOL  ; Actuele snelheid gelijk aan de wens snelheid
Com2_Alle_Oever_Poortjes_Gesloten 3332.15 BOOL  ; Alle Oever Poortjes zijn gesloten
Com2_Ingangs_Poortje_1_Links_Open 3332.01 BOOL
Com2_Open_Uitgangs_Poortjes 3333.03 BOOL  ; Open de Uitgangs Poortjes
Com2_Pulse 3337.03 BOOL
Com2_Sluit_Uitgangs_Poortjes_Oever 3333.04 BOOL  ; Sluit de Uitgangs Poortjes Oever
Com2_Vrijgave_Ingangs_Poortjes 3332.01 BOOL
DFACTOR_RANGE_1 D2851 CHANNEL
DFACTOR_RANGE_3 D2853 CHANNEL
DFACTOR_RANGE_5 D2855 CHANNEL
DFACTOR_RANGE_7 D2857 CHANNEL
D_Setpoint_1 D176 CHANNEL
M_ALM_1_1024 H164.00 BOOL  ; Alarm 1-0124 Er is minstens 1 alarm in de file Tourniquets
M_GROND_UITG_GESLOTEN W165.05 BOOL  ; GROND UITG GESLOTEN
M_Ingangs_Poortje_L_Dicht W160.02 BOOL
M_Ingangs_Poortjes_Links_Open W160.01 BOOL
M_Ingangs_Poortjes_R_Dicht W160.04 BOOL
M_Ingangs_Poortjes_R_Open W160.03 BOOL
M_Uitgangs_poortjes_Open W165.01 BOOL  ; Uitgangs Poortjes zijn Open
T_Sluit_Uitgangs_Poortjes T0166 BOOL  ; Maximale tijd sluit uitgangs poortjes
Totale_Dag_Teller_Tourniquets D159 CHANNEL  ; Totale Dag teller Linker & Rechter Tournoquets

### Section Tourniquets_Grond

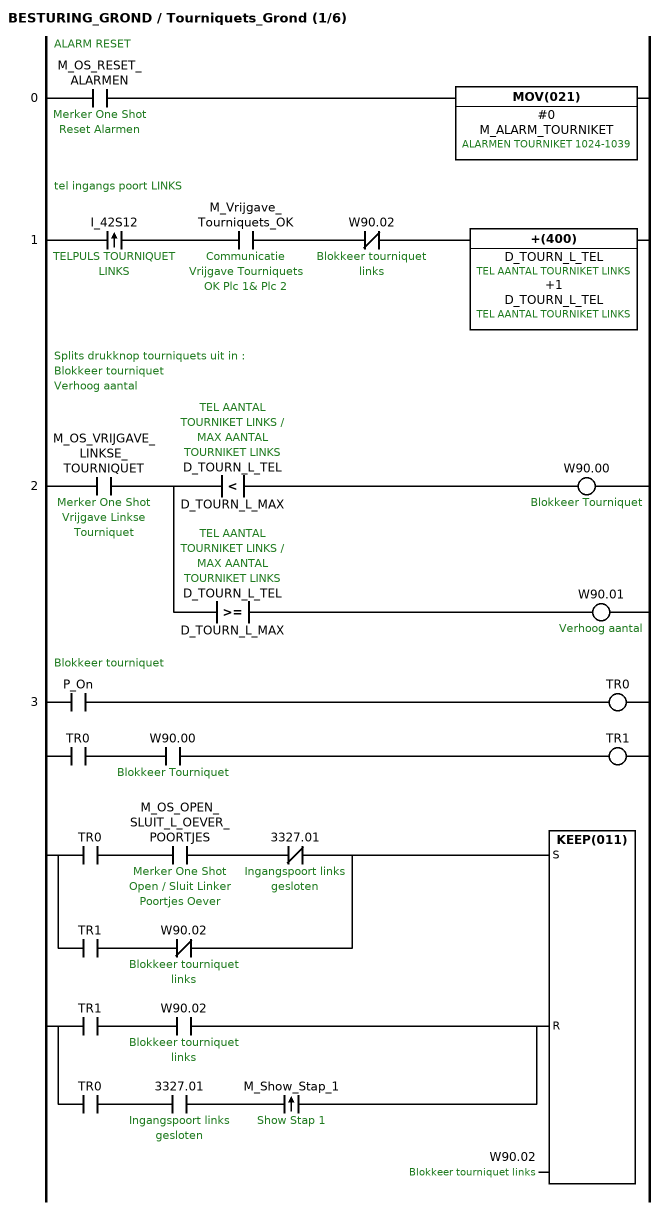
; rung 0: ALARM RESET
LD M_OS_RESET_ALARMEN  ; Merker One Shot Reset Alarmen
MOV(021) #0 M_ALARM_TOURNIKET  ; ALARMEN TOURNIKET 1024-1039
; rung 1: tel ingangs poort LINKS
@LD I_42S12  ; TELPULS TOURNIQUET LINKS
AND M_Vrijgave_Tourniquets_OK  ; Communicatie Vrijgave Tourniquets OK Plc 1& Plc 2
ANDNOT W90.02  ; Blokkeer tourniquet links
+(400) D_TOURN_L_TEL +1 D_TOURN_L_TEL  ; TEL AANTAL TOURNIKET LINKS
; rung 2: Splits drukknop tourniquets uit in : / Blokkeer tourniquet / Verhoog aantal
LD M_OS_VRIJGAVE_LINKSE_TOURNIQUET  ; Merker One Shot Vrijgave Linkse Tourniquet
OUT TR0
AND<(310) D_TOURN_L_TEL D_TOURN_L_MAX  ; TEL AANTAL TOURNIKET LINKS, MAX AANTAL TOURNIKET LINKS
OUT W90.00  ; Blokkeer Tourniquet
LD TR0
AND>=(325) D_TOURN_L_TEL D_TOURN_L_MAX  ; TEL AANTAL TOURNIKET LINKS, MAX AANTAL TOURNIKET LINKS
OUT W90.01  ; Verhoog aantal
; rung 3: Blokkeer tourniquet
LD P_On
OUT TR0
AND M_OS_OPEN_SLUIT_L_OEVER_POORTJES  ; Merker One Shot Open / Sluit Linker Poortjes Oever
ANDNOT 3327.01  ; Ingangspoort links gesloten
LD TR0
AND W90.00  ; Blokkeer Tourniquet
OUT TR1
ANDNOT W90.02  ; Blokkeer tourniquet links
ORLD
LD TR1
AND W90.02  ; Blokkeer tourniquet links
LD TR0
AND 3327.01  ; Ingangspoort links gesloten
@AND M_Show_Stap_1  ; Show Stap 1
ORLD
KEEP(011) W90.02  ; Blokkeer tourniquet links

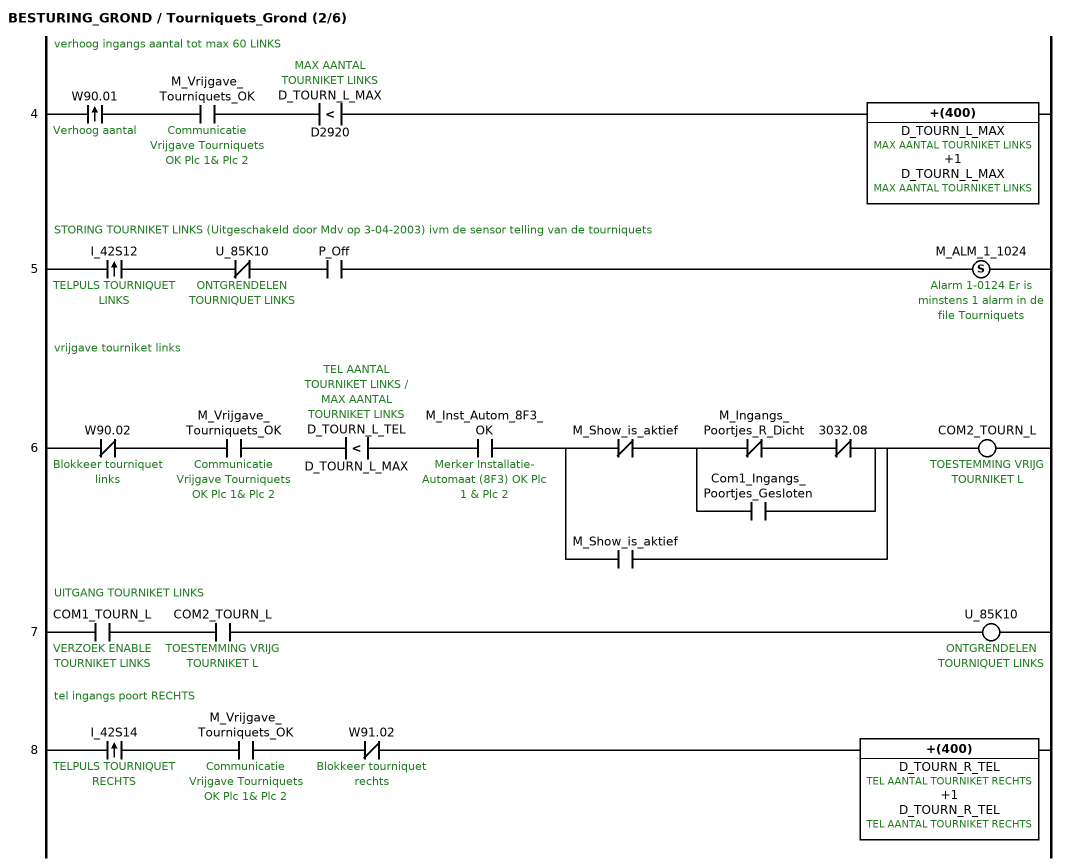
; rung 4: verhoog ingangs aantal tot max 60 LINKS
@LD W90.01  ; Verhoog aantal
AND M_Vrijgave_Tourniquets_OK  ; Communicatie Vrijgave Tourniquets OK Plc 1& Plc 2
AND<S(312) D_TOURN_L_MAX D2920  ; MAX AANTAL TOURNIKET LINKS
+(400) D_TOURN_L_MAX +1 D_TOURN_L_MAX  ; MAX AANTAL TOURNIKET LINKS
; rung 5: STORING TOURNIKET LINKS (Uitgeschakeld door Mdv op 3-04-2003) ivm de sensor telling van de tourniquets
@LD I_42S12  ; TELPULS TOURNIQUET LINKS
ANDNOT U_85K10  ; ONTGRENDELEN TOURNIQUET LINKS
AND P_Off
SET M_ALM_1_1024  ; Alarm 1-0124 Er is minstens 1 alarm in de file Tourniquets
; rung 6: vrijgave tourniket links
LDNOT W90.02  ; Blokkeer tourniquet links
AND M_Vrijgave_Tourniquets_OK  ; Communicatie Vrijgave Tourniquets OK Plc 1& Plc 2
AND<S(312) D_TOURN_L_TEL D_TOURN_L_MAX  ; TEL AANTAL TOURNIKET LINKS, MAX AANTAL TOURNIKET LINKS
AND M_Inst_Autom_8F3_OK  ; Merker Installatie-Automaat (8F3) OK Plc 1 & Plc 2
LDNOT M_Show_is_aktief
LDNOT M_Ingangs_Poortjes_R_Dicht
ANDNOT 3032.08
OR Com1_Ingangs_Poortjes_Gesloten
ANDLD
OR M_Show_is_aktief
ANDLD
OUT COM2_TOURN_L  ; TOESTEMMING VRIJG TOURNIKET L
; rung 7: UITGANG TOURNIKET LINKS
LD COM1_TOURN_L  ; VERZOEK ENABLE TOURNIKET LINKS
AND COM2_TOURN_L  ; TOESTEMMING VRIJG TOURNIKET L
OUT U_85K10  ; ONTGRENDELEN TOURNIQUET LINKS
; rung 8: tel ingangs poort RECHTS
@LD I_42S14  ; TELPULS TOURNIQUET RECHTS
AND M_Vrijgave_Tourniquets_OK  ; Communicatie Vrijgave Tourniquets OK Plc 1& Plc 2
ANDNOT W91.02  ; Blokkeer tourniquet rechts
+(400) D_TOURN_R_TEL +1 D_TOURN_R_TEL  ; TEL AANTAL TOURNIKET RECHTS

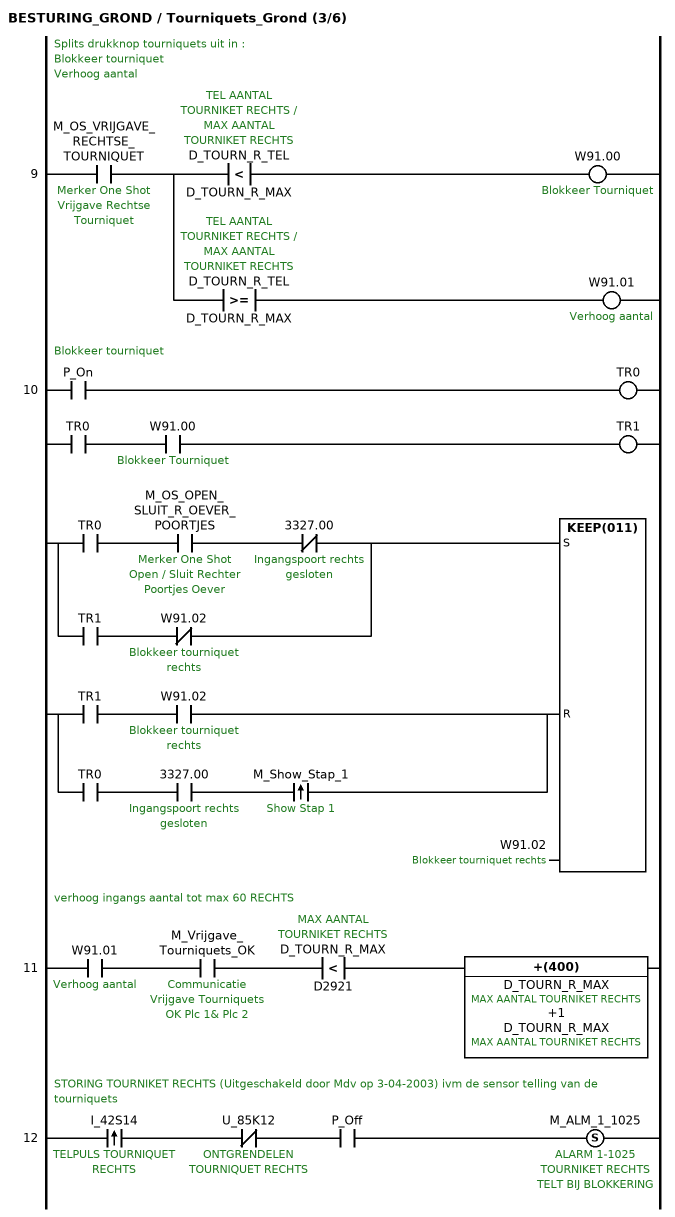
; rung 9: Splits drukknop tourniquets uit in : / Blokkeer tourniquet / Verhoog aantal
LD M_OS_VRIJGAVE_RECHTSE_TOURNIQUET  ; Merker One Shot Vrijgave Rechtse Tourniquet
OUT TR0
AND<(310) D_TOURN_R_TEL D_TOURN_R_MAX  ; TEL AANTAL TOURNIKET RECHTS, MAX AANTAL TOURNIKET RECHTS
OUT W91.00  ; Blokkeer Tourniquet
LD TR0
AND>=(325) D_TOURN_R_TEL D_TOURN_R_MAX  ; TEL AANTAL TOURNIKET RECHTS, MAX AANTAL TOURNIKET RECHTS
OUT W91.01  ; Verhoog aantal
; rung 10: Blokkeer tourniquet
LD P_On
OUT TR0
AND M_OS_OPEN_SLUIT_R_OEVER_POORTJES  ; Merker One Shot Open / Sluit Rechter Poortjes Oever
ANDNOT 3327.00  ; Ingangspoort rechts gesloten
LD TR0
AND W91.00  ; Blokkeer Tourniquet
OUT TR1
ANDNOT W91.02  ; Blokkeer tourniquet rechts
ORLD
LD TR1
AND W91.02  ; Blokkeer tourniquet rechts
LD TR0
AND 3327.00  ; Ingangspoort rechts gesloten
@AND M_Show_Stap_1  ; Show Stap 1
ORLD
KEEP(011) W91.02  ; Blokkeer tourniquet rechts
; rung 11: verhoog ingangs aantal tot max 60 RECHTS
LD W91.01  ; Verhoog aantal
AND M_Vrijgave_Tourniquets_OK  ; Communicatie Vrijgave Tourniquets OK Plc 1& Plc 2
AND<S(312) D_TOURN_R_MAX D2921  ; MAX AANTAL TOURNIKET RECHTS
+(400) D_TOURN_R_MAX +1 D_TOURN_R_MAX  ; MAX AANTAL TOURNIKET RECHTS
; rung 12: STORING TOURNIKET RECHTS (Uitgeschakeld door Mdv op 3-04-2003) ivm de sensor telling van de tourniquets
@LD I_42S14  ; TELPULS TOURNIQUET RECHTS
ANDNOT U_85K12  ; ONTGRENDELEN TOURNIQUET RECHTS
AND P_Off
SET M_ALM_1_1025  ; ALARM 1-1025 TOURNIKET RECHTS TELT BIJ BLOKKERING

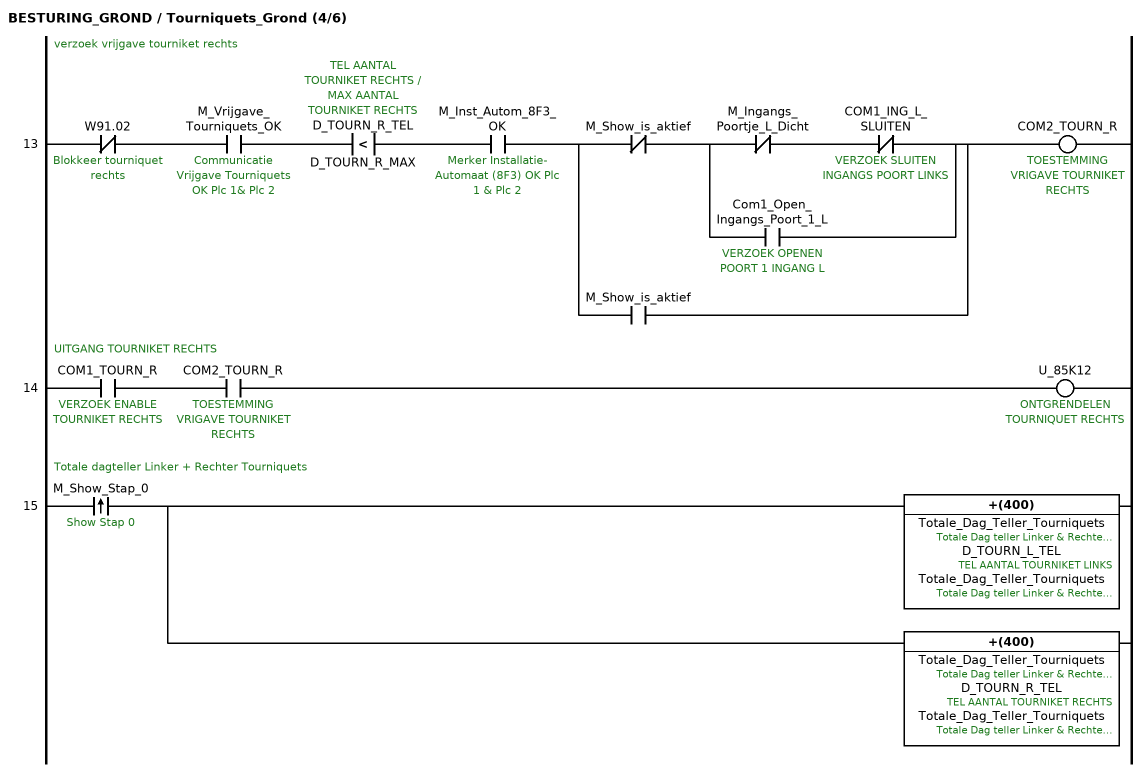
; rung 13: verzoek vrijgave tourniket rechts
LDNOT W91.02  ; Blokkeer tourniquet rechts
AND M_Vrijgave_Tourniquets_OK  ; Communicatie Vrijgave Tourniquets OK Plc 1& Plc 2
AND<S(312) D_TOURN_R_TEL D_TOURN_R_MAX  ; TEL AANTAL TOURNIKET RECHTS, MAX AANTAL TOURNIKET RECHTS
AND M_Inst_Autom_8F3_OK  ; Merker Installatie-Automaat (8F3) OK Plc 1 & Plc 2
LDNOT M_Show_is_aktief
LDNOT M_Ingangs_Poortje_L_Dicht
ANDNOT COM1_ING_L_SLUITEN  ; VERZOEK SLUITEN INGANGS POORT LINKS
OR Com1_Open_Ingangs_Poort_1_L  ; VERZOEK OPENEN POORT 1 INGANG L
ANDLD
OR M_Show_is_aktief
ANDLD
OUT COM2_TOURN_R  ; TOESTEMMING VRIGAVE TOURNIKET RECHTS
; rung 14: UITGANG TOURNIKET RECHTS
LD COM1_TOURN_R  ; VERZOEK ENABLE TOURNIKET RECHTS
AND COM2_TOURN_R  ; TOESTEMMING VRIGAVE TOURNIKET RECHTS
OUT U_85K12  ; ONTGRENDELEN TOURNIQUET RECHTS
; rung 15: Totale dagteller Linker + Rechter Tourniquets
@LD M_Show_Stap_0  ; Show Stap 0
+(400) Totale_Dag_Teller_Tourniquets D_TOURN_L_TEL Totale_Dag_Teller_Tourniquets  ; Totale Dag teller Linker & Rechter Tournoquets, TEL AANTAL TOURNIKET LINKS
+(400) Totale_Dag_Teller_Tourniquets D_TOURN_R_TEL Totale_Dag_Teller_Tourniquets  ; Totale Dag teller Linker & Rechter Tournoquets, TEL AANTAL TOURNIKET RECHTS

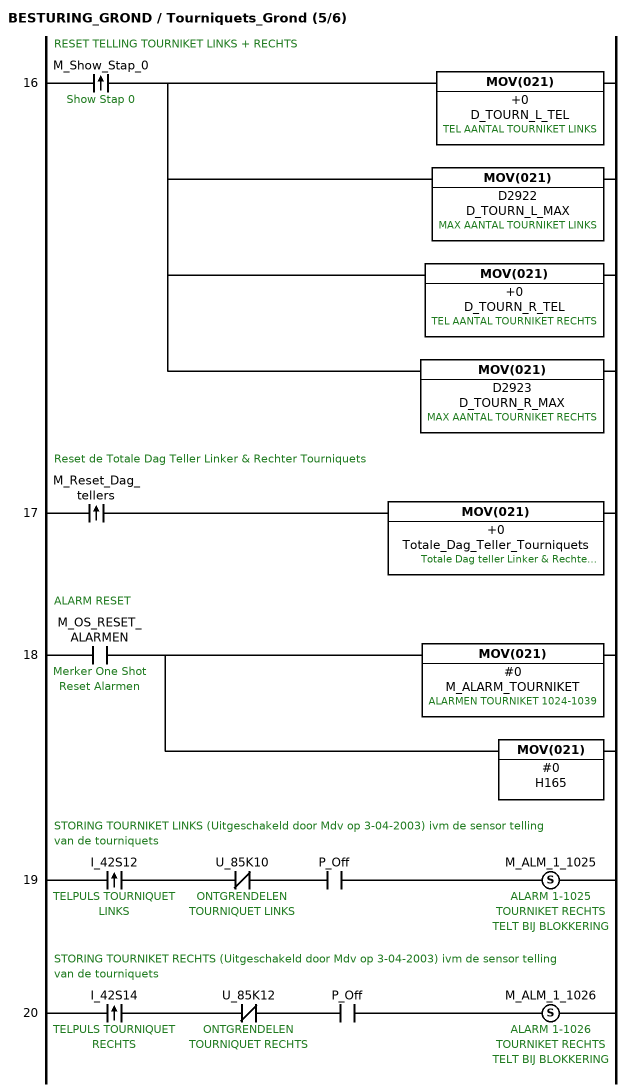
; rung 16: RESET TELLING TOURNIKET LINKS + RECHTS
@LD M_Show_Stap_0  ; Show Stap 0
MOV(021) +0 D_TOURN_L_TEL  ; TEL AANTAL TOURNIKET LINKS
MOV(021) D2922 D_TOURN_L_MAX  ; MAX AANTAL TOURNIKET LINKS
MOV(021) +0 D_TOURN_R_TEL  ; TEL AANTAL TOURNIKET RECHTS
MOV(021) D2923 D_TOURN_R_MAX  ; MAX AANTAL TOURNIKET RECHTS
; rung 17: Reset de Totale Dag Teller Linker & Rechter Tourniquets
@LD M_Reset_Dag_tellers
MOV(021) +0 Totale_Dag_Teller_Tourniquets  ; Totale Dag teller Linker & Rechter Tournoquets
; rung 18: ALARM RESET
LD M_OS_RESET_ALARMEN  ; Merker One Shot Reset Alarmen
MOV(021) #0 M_ALARM_TOURNIKET  ; ALARMEN TOURNIKET 1024-1039
MOV(021) #0 H165
; rung 19: STORING TOURNIKET LINKS (Uitgeschakeld door Mdv op 3-04-2003) ivm de sensor telling van de tourniquets
@LD I_42S12  ; TELPULS TOURNIQUET LINKS
ANDNOT U_85K10  ; ONTGRENDELEN TOURNIQUET LINKS
AND P_Off
SET M_ALM_1_1025  ; ALARM 1-1025 TOURNIKET RECHTS TELT BIJ BLOKKERING
; rung 20: STORING TOURNIKET RECHTS (Uitgeschakeld door Mdv op 3-04-2003) ivm de sensor telling van de tourniquets
@LD I_42S14  ; TELPULS TOURNIQUET RECHTS
ANDNOT U_85K12  ; ONTGRENDELEN TOURNIQUET RECHTS
AND P_Off
SET M_ALM_1_1026  ; ALARM 1-1026 TOURNIKET RECHTS TELT BIJ BLOKKERING

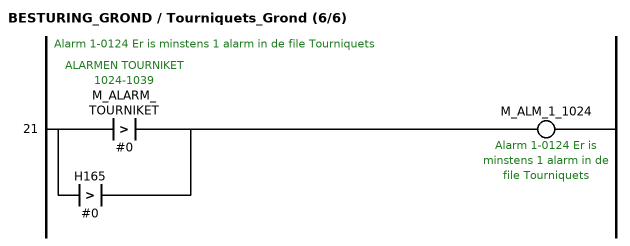
; rung 21: Alarm 1-0124 Er is minstens 1 alarm in de file Tourniquets
LD>(320) M_ALARM_TOURNIKET #0  ; ALARMEN TOURNIKET 1024-1039
OR>(320) H165 #0
OUT M_ALM_1_1024  ; Alarm 1-0124 Er is minstens 1 alarm in de file Tourniquets

### Section Ingangs_Poortjes_Grond

